// Mitsubishi GX Works2 project: 4. teaching_2   PLC: Q03UDV

PROGRAM MAIN
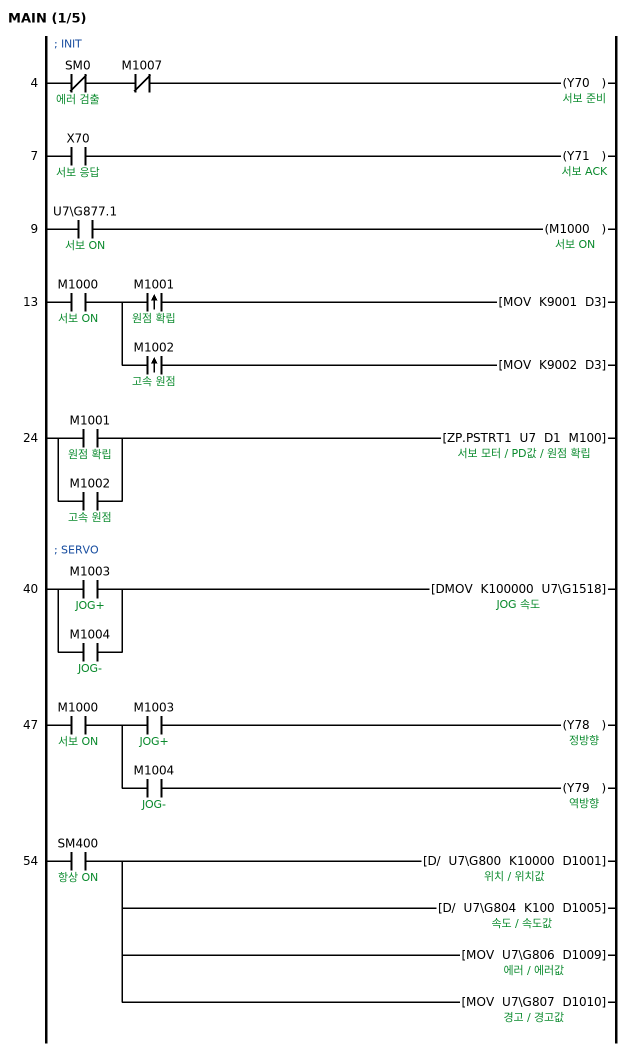
; INIT
4     LDI     SM0  ; 에러 검출
      ANI     M1007
      OUT     Y70  ; 서보 준비
7     LD      X70  ; 서보 응답
      OUT     Y71  ; 서보 ACK
9     LD      U7\G877.1  ; 서보 ON
      OUT     M1000  ; 서보 ON
13    LD      M1000  ; 서보 ON
      MPS
      ANDP    M1001  ; 원점 확립
      MOV     K9001 D3
      MPP
      ANDP    M1002  ; 고속 원점
      MOV     K9002 D3
24    LD      M1001  ; 원점 확립
      OR      M1002  ; 고속 원점
      ZP.PSTRT1 U7 D1 M100  ; 서보 모터 / PD값 / 원점 확립
; SERVO
40    LD      M1003  ; JOG+
      OR      M1004  ; JOG-
      DMOV    K100000 U7\G1518  ; JOG 속도
47    LD      M1000  ; 서보 ON
      MPS
      AND     M1003  ; JOG+
      OUT     Y78  ; 정방향
      MPP
      AND     M1004  ; JOG-
      OUT     Y79  ; 역방향
54    LD      SM400  ; 항상 ON
      D/      U7\G800 K10000 D1001  ; 위치 / 위치값
      D/      U7\G804 K100 D1005  ; 속도 / 속도값
      MOV     U7\G806 D1009  ; 에러 / 에러값
      MOV     U7\G807 D1010  ; 경고 / 경고값
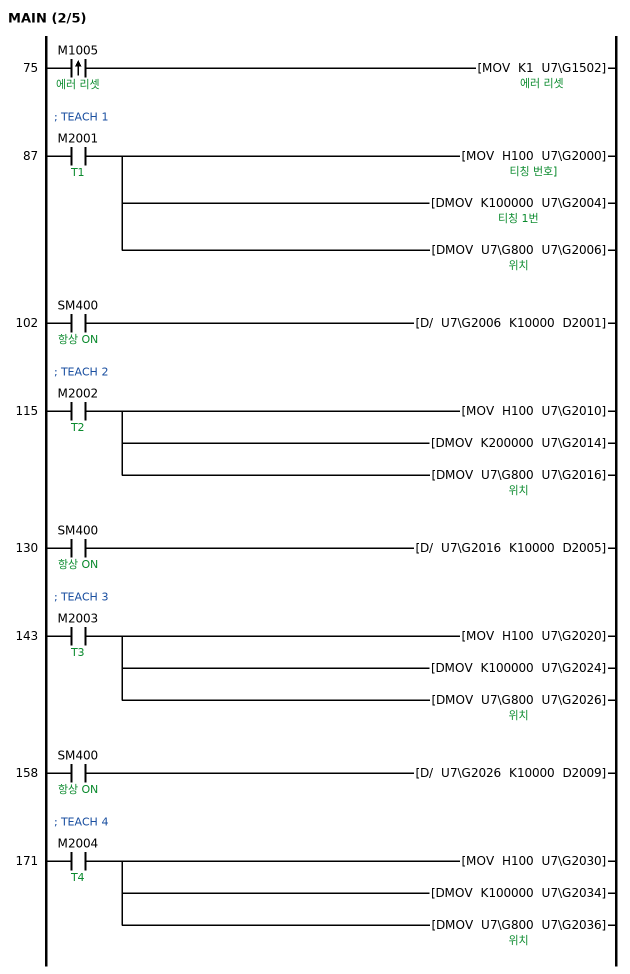
75    LDP     M1005  ; 에러 리셋
      MOV     K1 U7\G1502  ; 에러 리셋
; TEACH 1
87    LD      M2001  ; T1
      MOV     H100 U7\G2000  ; 티칭 번호]
      DMOV    K100000 U7\G2004  ; 티칭 1번
      DMOV    U7\G800 U7\G2006
102   LD      SM400  ; 항상 ON
      D/      U7\G2006 K10000 D2001
; TEACH 2
115   LD      M2002  ; T2
      MOV     H100 U7\G2010
      DMOV    K200000 U7\G2014
      DMOV    U7\G800 U7\G2016
130   LD      SM400  ; 항상 ON
      D/      U7\G2016 K10000 D2005
; TEACH 3
143   LD      M2003  ; T3
      MOV     H100 U7\G2020
      DMOV    K100000 U7\G2024
      DMOV    U7\G800 U7\G2026
158   LD      SM400  ; 항상 ON
      D/      U7\G2026 K10000 D2009
; TEACH 4
171   LD      M2004  ; T4
      MOV     H100 U7\G2030
      DMOV    K100000 U7\G2034
      DMOV    U7\G800 U7\G2036
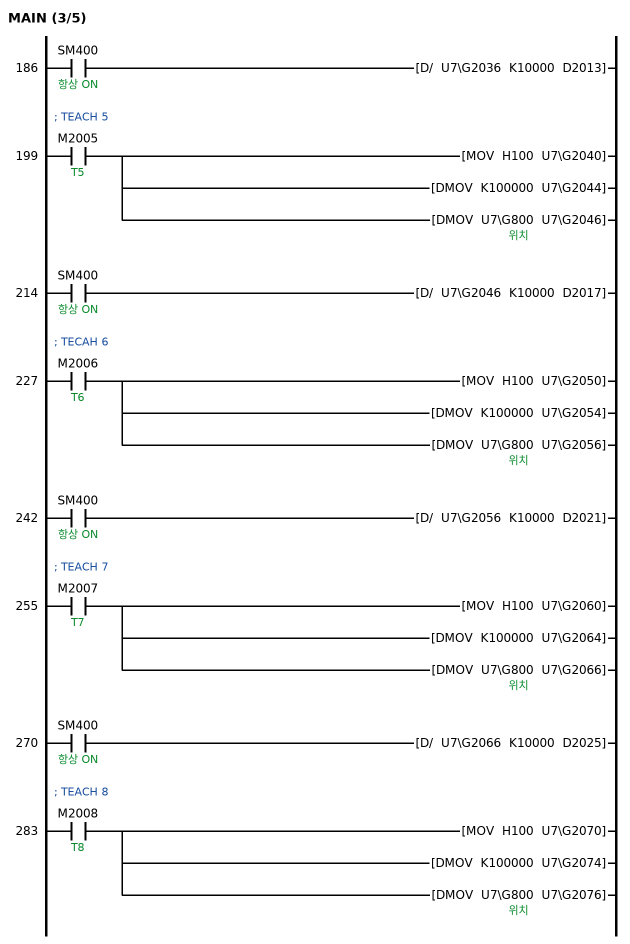
186   LD      SM400  ; 항상 ON
      D/      U7\G2036 K10000 D2013
; TEACH 5
199   LD      M2005  ; T5
      MOV     H100 U7\G2040
      DMOV    K100000 U7\G2044
      DMOV    U7\G800 U7\G2046
214   LD      SM400  ; 항상 ON
      D/      U7\G2046 K10000 D2017
; TECAH 6
227   LD      M2006  ; T6
      MOV     H100 U7\G2050
      DMOV    K100000 U7\G2054
      DMOV    U7\G800 U7\G2056
242   LD      SM400  ; 항상 ON
      D/      U7\G2056 K10000 D2021
; TEACH 7
255   LD      M2007  ; T7
      MOV     H100 U7\G2060
      DMOV    K100000 U7\G2064
      DMOV    U7\G800 U7\G2066
270   LD      SM400  ; 항상 ON
      D/      U7\G2066 K10000 D2025
; TEACH 8
283   LD      M2008  ; T8
      MOV     H100 U7\G2070
      DMOV    K100000 U7\G2074
      DMOV    U7\G800 U7\G2076
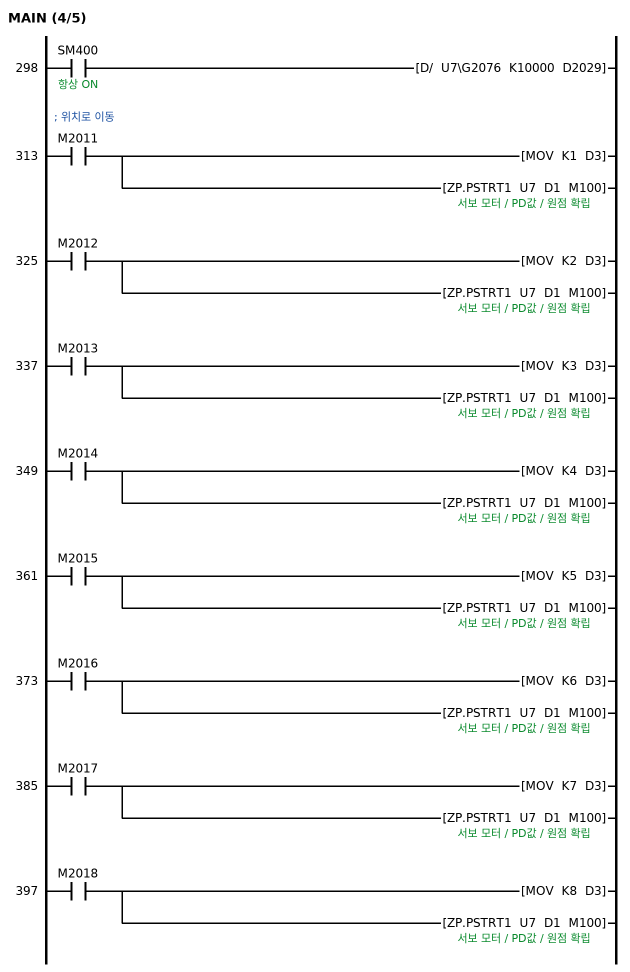
298   LD      SM400  ; 항상 ON
      D/      U7\G2076 K10000 D2029
; 위치로 이동
313   LD      M2011
      MOV     K1 D3
      ZP.PSTRT1 U7 D1 M100
325   LD      M2012
      MOV     K2 D3
      ZP.PSTRT1 U7 D1 M100
337   LD      M2013
      MOV     K3 D3
      ZP.PSTRT1 U7 D1 M100
349   LD      M2014
      MOV     K4 D3
      ZP.PSTRT1 U7 D1 M100
361   LD      M2015
      MOV     K5 D3
      ZP.PSTRT1 U7 D1 M100
373   LD      M2016
      MOV     K6 D3
      ZP.PSTRT1 U7 D1 M100
385   LD      M2017
      MOV     K7 D3
      ZP.PSTRT1 U7 D1 M100
397   LD      M2018
      MOV     K8 D3
      ZP.PSTRT1 U7 D1 M100
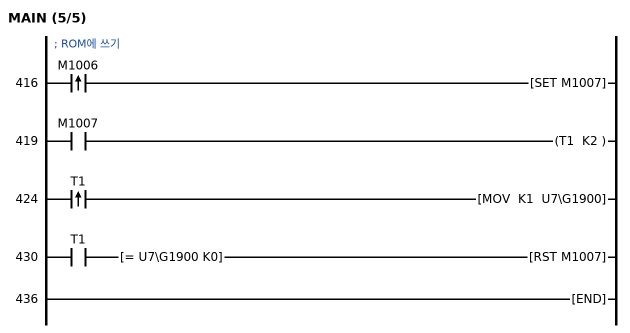
; ROM에 쓰기
416   LDP     M1006
      SET     M1007
419   LD      M1007
      OUT     T1 K2
424   LDP     T1
      MOV     K1 U7\G1900
430   LD      T1
      AND=    U7\G1900 K0
      RST     M1007
436   END
END_PROGRAM

// device comments not shown above
X0  ; 공급 후진
X1  ; 공급 전진
X2  ; 분배 후진
X3  ; 분배 전진
X4  ; 가공 상승
X15  ; PB1
X16  ; PB2
X17  ; PB3
X1C  ; Toggle
Y20  ; 공급+
Y21  ; 공급-
Y22  ; 분배+
Y23  ; 분배-
M1  ; 공급+
M2  ; 공급-
M3  ; 분배+
M4  ; 분배-
M10  ; 무한 반복
P1  ; STOP
